TYPE EtcSlaveBase_82538BE2 :
STRUCT
END_STRUCT
END_TYPE

(* stored: Version 1.2.0.0, ProductVersion 3.1.4024.9
   DUT EtcSlaveBase_82538BE2: Id {011fe121-fa97-4f1b-866b-928ddbf3f692} *)
